PROGRAM MAIN
VAR
	FB_Control1: FB_Control;
	FB_Motion1: FB_Motion;

END_VAR



FB_Control1(button1:=binput1 , ProcessDone:=main.FB_Motion1.bDone , ProgEx=> );

FB_Motion1(
	bStart:=binput1 , 
	bExecute:=main.FB_Control1.ProgEx , 
	bBusy=> , 
	bDone=> , 
	nPosition:=main.FB_Control1.position , 
	);

END_PROGRAM

(* stored: Version 1.1.0.1, ProductVersion 3.1.4022.16
   POU MAIN: Id {b1e4c4d8-fc6f-41a6-9419-ff9372b5a71d}, SpecialFunc None *)
